TYPE ST_HMI_DataSourceConfig : 
STRUCT
	nID: DINT;
	sDisplayName: WSTRING(80);
	eConfigType: E_SourceType;
	aInputSources: ARRAY [0..0] OF ST_HMI_InputSource;
END_STRUCT
END_TYPE

(* stored: DUT ST_HMI_DataSourceConfig: Id a86d051b-7fbb-429a-bbbf-809139eee1b1 *)
